// TwinCAT 3 PLC project AMKO_System
// Title: IBF_System
// Company: Industrial Brains B.V.
// ProjectVersion: 0.0.0.0
// Description: system and module base functions
// ProgramVersion: 3.1.4023.0
// libraries:
//   Device_Library, * (AMKO-Engineering)
//   HMI_Library, * (AMKO-Engineering)
//   Tc2_Standard, * (Beckhoff Automation GmbH)
//   Tc2_System, * (Beckhoff Automation GmbH)
//   Tc2_Utilities, * (Beckhoff Automation GmbH)
//   Tc3_Module, * (Beckhoff Automation GmbH)
//   Utilities_Library, * (AMKO-Engineering)
// project tree:
//   / PlcTask.TcTTO
//   FaultHandler/ Fb_SystemFaultHandler.TcPOU
//   GVLs/ GVL_Main.TcGVL
//   ModuleBase/Base/ Fb_ModuleBase.TcPOU
//   ModuleBase/DataTypes/ Udt_ModuleBase.TcDUT
//   SystemBase/DataTypes/ E_StateSystem.TcTLEO, Udt_ModuleId.TcDUT (not stored)
//   SystemBase/ SystemBase.TcPOU
//   _TESTS/ FB_DummyModule.TcPOU, PRG_TEST.TcPOU

CONFIGURATION AMKO_System
    RESOURCE PLC ON TwinCAT3
        TASK PlcTask(INTERVAL := T#10ms, PRIORITY := 20);
        PROGRAM SystemBase WITH PlcTask : SystemBase;
    END_RESOURCE
END_CONFIGURATION

// ---- ModuleBase/DataTypes/Udt_ModuleBase.TcDUT
TYPE Udt_ModuleBase :
STRUCT
	sModuleName 		: STRING := 'NA' 		; // Module name
	bModuleActive		: 	BOOL := FALSE 		; // Module is active in the system (will be ignored by system if false) 	
	// safety Inputs
	bEstopOk			:	BOOL ; // When estop is not ok, complete machine is shut down and reinitialization is required.
	bModuleSafetyOk		: 	BOOL ; // Module safety systems are ok and safe 
	bAirPressureOk		: 	BOOL ; // system safety condition monitorring air pressure ok
	bPowerSupplyOk		: 	BOOL ; // System power supply is ok
	// main system Inputs
	bCmdStart			: 	BOOL	:= FALSE ; // System start command 
	bCmdReset 			: 	BOOL	:= FALSE ; // reset all faults 
	bCmdPowerOff		:	BOOL	:= FALSE ; // power off module 
	bCmdStartManual 	: 	BOOL 	:= FALSE ; // Start up in manual mode
 	// Com to main system
	fbFaultHandler		: 	Fb_FaultHandler 		; // Fault handler 
	sStateIndicator		: 	STRING := ''			; // Operator message, indication of current step or function 

	// Fault indications
	bMissingCond	: BOOL := FALSE ; // Module missing condition active
	bFatalFault		: BOOL := FALSE ; // Module fatal fault is active
	bCycleFault		: BOOL := FALSE ; // Module cycle fault is active
	bOperatorWarning : BOOL := FALSE; //

	// State indication
	bIsSafe			: BOOL := FALSE ; // Module is safe and locked until safety is ok
	bNoreference	: BOOL := FALSE ; // Module Startup Undefined initialization required

	bInitializing	: BOOL := FALSE ; // Module startup initializing
	bInitialized	: BOOL := FALSE ; // Module startup initialized waiting for startup command

	bIdle 			: BOOL := FALSE ; // Module startup Idle no commands active

	bEnabling 		: BOOL := FALSE ; // Module Startup enabeling 
	bEnabled 		: BOOL := FALSE ; // Module Startup Enabled
	
	bHoming			: BOOL := FALSE ; // Module startup homing back to base position and recalibrate
	bHomed 			: BOOL := FALSE ; // Module startup homed waiting for further further commands

	bHolding 		: BOOL := FALSE ; // Module Module Hold motion command executing
	bHeld	 		: BOOL := FALSE ; // Module Hold Motion is held until command is released	
	
	bResetting 		: BOOL := FALSE ; // Module Reset resetting error status
	bResetDone 		: BOOL := FALSE ; // Module reset is done   

	bManual 		: BOOL := FALSE ; // Module Work status Module in Manual 
	bAutomatic 		: BOOL := FALSE ; // Module Work status Module in Automatic mode
	
	bPoweringOff	: BOOL := FALSE ; // Module is powering off
	bPoweredOff		: BOOL := FALSE ; // Module has powered off 	
	
	// manual functions 
	bDevicesAddedtoManual	: BOOL := FALSE ;
	bParametersAdded		: BOOL := FALSE ;
	// Persistent data
	bCmdWritePersistent  : BOOL := false ; // write persistent data to memory
END_STRUCT
END_TYPE

// ---- SystemBase/DataTypes/E_StateSystem.TcTLEO
{attribute 'qualified_only'}
{attribute 'strict'}
{attribute 'to_string'}
TYPE E_StateSystem :
(
	NoReference		, 	// system has not been initialized
	Initialize		, 	// System is initializing
	LoadParameters	, 	// System is loading parameters from/to file
	Safe			, 	// System is in safety state
	Enable			, 	// System is enabling 
	Home			, 	// system is hominig 
	Resetting		, 	// System is resetting
	Idle			, 	// system is waiting for commands
	Manual			, 	// System is in manual mode
	SemiAuto		, 	// System is in semi auto mode
	Automatic		, 	// system is in automatic mode 
	Fault			,	// System is in Fault state
	PowerOff		// system is powering off
)INT;
END_TYPE

// ---- GVLs/GVL_Main.TcGVL

{attribute 'qualified_only'} // Main system variables and state indicators
{attribute 'analysis':= '-33'}
VAR_GLOBAL CONSTANT
	cnMaxNUMBEROFMODULES 	: UDINT := 10 		; // "maximum" number of modules in the system
	CtAIRPRESSUREDELAY	: TIME 	:= T#500MS	; // Timout before air fault becomes active
	cbUPSPRESENT		: BOOL	:= FALSE 	; // Enable automatic shutdown when power is interupted
END_VAR
VAR_GLOBAL PERSISTENT
	nTotalUnitsProduced		: UDINT ; // Units produced 
END_VAR

// ---- SystemBase/SystemBase.TcPOU
{attribute 'reflection'}
PROGRAM SystemBase // system base program, from here all modules are controlled and the system functions are called.
VAR_INPUT // System configuration settings
	bIcfAirCheckPresent	: BOOL := TRUE; // System is not equiped with air pressure sensor 
END_VAR
VAR	// Fault indications
	bMissingCond		: BOOL := FALSE ; // Module missing condition active
	bFatalFault			: BOOL := FALSE ; // Module fatal fault is active
	bCycleFault			: BOOL := FALSE ; // Module cycle fault is active
	bOperatorWarning	: BOOL := FALSE ; // Module operator warning is active

	// Check values
	bReferenceOk		: BOOL := FALSE ; // All module references  have been checked

	// State indication
	bSafeStopping		: BOOL := FALSE ; // Module is stopping by safety
	bIsSafe				: BOOL := FALSE ; // Module is safe and locked until safety is ok
	bNoreference		: BOOL := FALSE ; // Module Startup Undefined initialization required

	bInitializing		: BOOL := FALSE ; // Module startup initializing
	bInitialized		: BOOL := FALSE ; // Module startup initialized waiting for startup command
	
	bParametersLoaded 	: BOOL := FALSE ; // Parameters have been loaded from the file(s) 

	bIdle 				: BOOL := FALSE ; // Module startup Idle no commands active

	bEnabling 			: BOOL := FALSE ; // Module Startup enabeling 
	bEnabled 			: BOOL := FALSE ; // Module Startup Enabled
	
	bHoming				: BOOL := FALSE ; // Module startup homing back to base position and recalibrate
	bHomed 				: BOOL := FALSE ; // Module startup homed waiting for further further commands

	bHolding 			: BOOL := FALSE ; // Module Module Hold motion command executing
	bHeld	 			: BOOL := FALSE ; // Module Hold Motion is held until command is released	
	
	bResetting 			: BOOL := FALSE ; // Module Reset resetting error status
	bResetDone 			: BOOL := FALSE ; // Module reset is done   

	bManual 			: BOOL := FALSE ; // Module Work status Module in Manual 
	
	bStartSemiAuto		: BOOL := FALSE ; // Start semi automatic mode 
	bSemiAuto			: BOOL := FALSE ; // Module work status module in semi automatic
	
	bStartAuto			: BOOL := FALSE ; // Start automatic mode
	bAutomatic 			: BOOL := FALSE ; // Module Work status Module in Automatic mode
	bStopAuto			: BOOL := FALSE ; // Start automatic mode
	bStoppingAuto		: BOOL := FALSE ; // Start automatic mode
	
	bCmdPause			: BOOL := FALSE ; // Pause all modules 
	bPaused 			: BOOL := FALSE ; // all modules are paused
	
	bPoweringOff		: BOOL := FALSE ; // Module is powering off
	bPoweredOff			: BOOL := FALSE ; // Module has powered off 	

	bModuleLocked		: BOOL := FALSE ; // a module is locked for commands
	
	bAckWarningsBusy	: BOOL := FALSE	; // The acknowledge process is busy
END_VAR
VAR
	// System inputs 
	ibPowerSupplyOk	 	AT%I*	: BOOL  ; // System Power supply is ok 
	iSystemSafetyFault	AT%I*	: BOOL	; // System safety Fault
	fbAirpressureOk 			: Fb_DevDigitalInputFunctions  	; // system airpressure is ok
	fbCmdResetSafety		 	: FB_DevPushbuttonLight 		; // System reset
	
	fTrigPowerSupply			: F_TRIG ; // falling edge trigger for power supply
	toffMainAir					: TOF	:= (PT := T#500MS ); // Main air supply off delay
	// System safety valve
	fbValveMainAirSupply		: FB_DevValve ; // Main air supply valve 
	
	// System HMI commands
	fbStartSemiAuto				: FB_DevHMIButton ; // HMI start semi automatic button 
	fbStartAuto					: FB_DevHMIButton ; // HMI start automatic button
	fbResetSystem				: FB_DevHMIButton ; // HMI Reset system
	fbCmdPowerOff				: FB_DevHMIButton ; // HMI Power off system
	fbAckWarning				: FB_DevHMIButton ; // HMI Acknowledge warnings

	// system Commands 
	fbCmdStartSystem		 	: FB_DevPushbuttonLight  		; // (re)start system input from button
	fbCmdStartAuto				: FB_DevPushbuttonLight			; // Start system automatic cycle
	fbCmdStopAuto				: FB_DevPushbuttonLight			; // Start system automatic cycle
	
	//System state
	bSafetyOK					: BOOL := FALSE ;
	bAirOk						: BOOL := FALSE ; // Air pressure is ok 
	bSystemOK					: BOOL := FALSE ; // all safety and vitals are OK
	eStateSystem				: E_StateSystem := E_StateSystem.NoReference ; // State of system
	// Set system variables
	fbSetSystemVariables		: Fb_SystemVariables ;
	
	// System Fault handling
	fbSystemFaultHandler		: Fb_SystemFaultHandler ;
	fbOperatorMessage			: FB_OperatorMessageDisplay ; //Operator message or system state message hadler 

	// Local Fault Handling
	fbFaultHandler				: Fb_FaultHandler 		; // Fault handler 
	stMessage					: UDT_Fault			; // Message data

 	// Module states
	nNumberOfModules			: UDINT := 0 ; // Number of modules added to the system 
	arpModules					: ARRAY [1..gvl_main.cnMaxNUMBEROFMODULES] OF Udt_ModuleId ; 

	// power down system function
	ntShutDown					: NT_Shutdown ; // shutdown system function 

	// Manual controller
	bDevicesAddedtoManual 		: BOOL := FALSE ; // Add system device (buttons) to manual controller
	

	// Function path 
	{attribute 'instance-path'} 
    {attribute 'noinit'}
	sPath			: STRING	; // Path name of function (used for manual reference
END_VAR
VAR // safety 
	// inputs 
	ibEstopOk 			AT%I*	: BOOL  ; // system emergency stop ok
	ibSystemSafetyOK	AT%I*	: BOOL  ; // System is safe 
	iSafetyFBErr		AT%I*	: BOOL	; // The "FB Error" group signal
	iSafetyComErr		AT%I*	: BOOL	; // The "Com Error" group signal
	iSafetyOtherErr		AT%I*	: BOOL	; // The "Other Err" group signal
	iSafetyOutErr		AT%I*	: BOOL	; // The "Out Err" group signal
	iSTOFault			AT%I* 	: BOOL	; // Motor safe torque off fault active
	
	// Outputs 
	qbSafetyErrAckn		AT%Q*	: BOOL ; // Safety error acknowledge
	qbRunSafety			AT%Q*	: BOOL ; // Run safety program
	qbResetSafety		AT%Q*	: BOOL ; // reset safety program
	qbSTOErrAckn		AT%Q*	: BOOL ; // Safet torque off error acnowledge

	// safety Reset Timer	
	TofSafetyErrAck				: TOF := (PT := T#500MS); // Safety reset timer
	TOfSTOErrAck				: TOF := (PT := T#500MS); // Safe torque off rest timer
END_VAR
VAR // Miscellaneous
	bFirstCycle : BOOL := TRUE; // Is this the first time the PRG is called?
	bPersistentDataFail	: BOOL := TRUE ;
END_VAR
VAR PERSISTENT // Persistent data check
	bPersistentFlag	: BOOL := FALSE ; // Persistent dat in tack flag
END_VAR

// Exec safety control
ExecSafetyControl();

// Call faulthandler
fbSystemFaultHandler( 	nNumberOfModules	:= nNumberOfModules,
						arpModules			:= arpModules,
						bsystemInitialized	:= bInitialized,
						bSystemFF			=> bFatalFault,
						bSystemCF			=> bCycleFault,
						bSystemMC			=> bMissingCond,
						bSystemOW			=> bOperatorWarning);

// Check if this is the first cycle the PRG is called
// if not, return. This is to make sure all modules are connected. 
IF bFirstCycle THEN
	bFirstCycle := FALSE;
	RETURN;
END_IF

// check system functions
IF bInitialized AND bParametersLoaded THEN 
	CheckSystemOK();
	CheckSystemCommands();
END_IF 

// Run system
ExecSystemRun();

// call device functions 
CallSystemFunctions();

// Call operator warning acknowledgement
ExecAckWarnings();

// Call modules 
CallModules();

METHOD PRIVATE CallModules : BOOL
VAR
	i : UDINT ;
END_VAR
VAR
	AllAutomatic : BOOL ;
	
	Stopping : BOOL;
	bAllStopped : BOOL;
END_VAR
// set base conditions
bReferenceOk	:= TRUE ;
bIsSafe			:= TRUE ;
bIdle			:= TRUE ;	
bHeld			:= TRUE ;
bResetDone 		S= bResetting	;
bManual			:= TRUE	;
bSemiAuto		:= TRUE ;
bAutomatic		:= FALSE; // Reverse feedback 
AllAutomatic 	:= TRUE ;
bStoppingAuto	:= TRUE ;
bEnabled		S= bEnabling ;
bPoweredOff		:= TRUE;
bHomed 			:= TRUE;
bPaused 		:= TRUE;
bAllStopped     := TRUE;

// copy inputs to modules 
FOR i := 1 TO nNumberOfModules DO 
	// set system commands
	arpModules[i].pFunction^.bEnable			:= bEnabled			;
	arpModules[i].pFunction^.bCmdReset			:= bResetting		;
	arpModules[i].pFunction^.bSafetyOK			:= NOT bSafeStopping;
	arpModules[i].pFunction^.bCmdPause			:= bCmdPause		; 
	// Read state indications 
	bReferenceOk 	:= arpModules[i].pFunction^.bReferenceOk 	AND bReferenceOk; 
	bIsSafe 		:= arpModules[i].pFunction^.bIsSafe 		AND bIsSafe		;
	bEnabled 		:= arpModules[i].pFunction^.bEnable 		AND bEnabled	;
	bHeld			:= arpModules[i].pFunction^.bHeld 			AND bHeld		;
	bResetDone		:= arpModules[i].pFunction^.bResetDone 		AND bResetDone	;
	bManual			:= arpModules[i].pFunction^.bManual 		AND bManual		;
	bSemiAuto		:= arpModules[i].pFunction^.bSemiAuto 		AND bSemiAuto	;
	bPoweredOff 		:= arpModules[i].pFunction^.bPoweredOff 		AND bPoweredOff	;
	bHomed			:= arpModules[i].pFunction^.bHomed			AND bHomed 		;
	bPaused			:= arpModules[i].pFunction^.bPaused			AND bPaused		;
	bModuleLocked	S= arpModules[i].pFunction^.bLocked							; // Module is locked for commnds
	bCmdPause 		R= arpModules[i].pFunction^.bReqContinue					; // Request continue from module
	bCmdPause		S= arpModules[i].pFunction^.bReqPause						; // Request for pause from module
	bAutomatic		S= arpModules[i].pFunction^.bAutomatic 						; // Stay in automatic even when one module is in automatic
	AllAutomatic	:= arpModules[i].pFunction^.bAutomatic 		AND AllAutomatic; // reset start automatic when al modules are in automatic operation
	bStoppingAuto	:= arpModules[i].pFunction^.bStopping 		AND bStoppingAuto; // reset start automatic when al modules are in automatic operation

	Stopping		:= arpModules[i].pFunction^.bStopping;
	
	bAllStopped     := NOT Stopping AND NOT bAutomatic AND bAllStopped;

	
END_FOR

// Reset start inputs
	bEnabling		R= bEnabled 	;
	bHolding		R= bHeld 		;
	bResetting		R= bResetDone 	;
	bStartSemiAuto	R= bSemiAuto	;
	bPoweringOff	R= bPoweredOff 	;
	bHoming			R= bHomed 		;
	bStartAuto		R= AllAutomatic	; 
	bStopAuto		R= bAllStopped	;
	bCmdPause		R= NOT bAutomatic	;
END_METHOD

METHOD PRIVATE CallSystemFunctions : BOOL
VAR_INPUT
END_VAR
// call parameter handler
GVL_Parameters.fbParameterHandler();
Device_Library.GVL_DevManual.fbManualControler();

// Execute button functions 
fbStartAuto		( 	tDelay			:= T#100MS,
					refFbManualCtrl	:= Device_Library.GVL_DevManual.fbManualControler,
					refFbFault 		:= fbFaultHandler );
fbStartSemiAuto ( 	tDelay			:= T#100MS,
					refFbManualCtrl	:= Device_Library.GVL_DevManual.fbManualControler,
					refFbFault 		:= fbFaultHandler ); 
fbResetSystem 	( 	Istatus			:= GVL_Message.bResetFaults,
					tDelay			:= T#5000MS,
					refFbManualCtrl	:= Device_Library.GVL_DevManual.fbManualControler,
					refFbFault 		:= fbFaultHandler ); 
fbAckWarning	(	Istatus			:= GVL_Message.bAckWarnings,
					tDelay			:= T#100MS,
					refFbManualCtrl := Device_Library.GVL_DevManual.fbManualControler,
					refFbFault 		:= fbFaultHandler );

fbCmdStartSystem(	refFbManualCtrl	:= Device_Library.GVL_DevManual.fbManualControler,
					refFbFault 		:= fbFaultHandler);
fbCmdStartAuto	(	refFbManualCtrl	:= Device_Library.GVL_DevManual.fbManualControler,
					refFbFault 		:= fbFaultHandler);
fbCmdStopAuto	(	refFbManualCtrl	:= Device_Library.GVL_DevManual.fbManualControler,
					refFbFault 		:= fbFaultHandler);

// execute input functions
fbValveMainAirSupply(	bEnable			:= TRUE,
						bSafetyOk		:= ibEstopOk,
						refFbManualCtrl	:= Device_Library.GVL_DevManual.fbManualControler,
						refFbFault 		:= fbFaultHandler);

// Add device functions to manual controller 
IF NOT bDevicesAddedtoManual THEN
	IF bIcfAirCheckPresent THEN
		Device_Library.GVL_DevManual.fbManualControler.CmdAddDevice( refToDevice := fbAirpressureOk 	);
	END_IF
	Device_Library.GVL_DevManual.fbManualControler.CmdAddDevice( refToDevice := fbCmdStartSystem	);
	Device_Library.GVL_DevManual.fbManualControler.CmdAddDevice( refToDevice := fbCmdStartAuto		);
	Device_Library.GVL_DevManual.fbManualControler.CmdAddDevice( refToDevice := fbCmdStopAuto		);
	Device_Library.GVL_DevManual.fbManualControler.CmdAddDevice( refToDevice := fbCmdResetSafety	);
	bDevicesAddedtoManual S= TRUE ;
END_IF
END_METHOD

METHOD INTERNAL CheckSystemCommands : BOOL
VAR_INPUT
END_VAR
// ===== full reset ======
	IF fbCmdResetSafety.bFcoDelay THEN 
		eStateSystem 	:= E_StateSystem.NoReference ;
	END_IF

// ====== power off ======
	IF fbCmdPowerOff.bFcoDelay THEN 
		eStateSystem := E_StateSystem.PowerOff ;
	END_IF
END_METHOD

METHOD PRIVATE CheckSystemOK : BOOL
// shutdown emediately if power is down 
fTrigPowerSupply(CLK := ibPowerSupplyOk);
ntShutDown(START := GVL_Main.cbUPSPRESENT AND (bPoweredOff OR fTrigPowerSupply.Q)); 

// ===== Check Air pressure =====
IF bIcfAirCheckPresent THEN
	fbAirpressureOk(refFbManualCtrl	:= Device_Library.GVL_DevManual.fbManualControler,
					refFbFault 		:= fbFaultHandler);
	bAirOk := fbAirpressureOk.bFcoDelay ;
ELSE
	bAirOk := TRUE ;
END_IF


// ===== Check if system is ok =====
	bSystemOK := TRUE ;
	bSystemOK := bAirOk 	AND bSystemOK ;
	bSystemOK := bSafetyOK	AND bSystemOK ;	
				
	IF NOT bSystemOK 
	AND eStateSystem > E_StateSystem.Safe 
	AND eStateSystem <> E_StateSystem.Resetting 
	THEN
		eStateSystem := E_StateSystem.Safe; 
	ELSIF (bFatalFault OR bCycleFault) 
	AND eStateSystem <> E_StateSystem.Resetting 
	THEN 
		eStateSystem := E_StateSystem.Fault ;
	END_IF

// ===== release system stop =====
bSafeStopping 	R= bIsSafe AND bSystemOK 		;
	
// ===== System messages ======
	IF NOT bAirOk THEN
		stMessage.Active 		:= TRUE ;
		stMessage.ComponentType	:= E_ComponentTypes.SafeIO ;
		stMessage.Discription	:= 'Main air Pressure low ';
		stMessage.LocationName	:= 'Main air supply';
		stMessage.LocationNumber:= 1;
		stMessage.FaultType		:= Utilities_Library.E_FaultTypes.FF;
		stMessage.MessageNumber	:= E_MessageNumbers.FF_Overload;
		stMessage.nModuleID		:= 0;
		GVL_HMI.bEstopActive 	:= TRUE ;
		GVL_HMI.sCmdEstopText 	:= 'AIR PRESSURE LOW';
	END_IF
	
// Main air control 
toffMainAir(IN := bSystemOK);
IF toffMainAir.Q THEN
	fbValveMainAirSupply.CmdOpen();
END_IF
END_METHOD

METHOD PUBLIC CmdAddModule : BOOL
VAR_INPUT
	refToModule : REFERENCE TO Fb_ModuleBase ; // reference to module function
END_VAR
VAR
	bModuleAdded	: BOOL := FALSE;
	i 				: UDINT ; 
END_VAR
// Check if device is not already in the array 
FOR i:= 1 TO GVL_Main.cnMaxNUMBEROFMODULES DO
	IF arpModules[i].pFunction = 0 THEN 
		nNumberOfModules:= i;
		EXIT;	
	ELSIF arpModules[i].sName = refToModule.sName THEN 
		bModuleAdded := TRUE ;
	END_IF 
END_FOR

// If device is not found add device to the list
IF NOT bModuleAdded AND nNumberOfModules >= 1 AND nNumberOfModules <= GVL_Main.cnMaxNUMBEROFMODULES THEN
	arpModules[nNumberOfModules].nNumber 	:= refToModule.nModuleID;
	arpModules[nNumberOfModules].sName		:= refToModule.sName	;
	arpModules[nNumberOfModules].pFunction 	:= ADR(refToModule)		;	
	bModuleAdded := TRUE ;
END_IF

CmdAddModule := bModuleAdded ;
END_METHOD

METHOD CmdReset : BOOL
VAR_INPUT
END_VAR
eStateSystem := E_StateSystem.Resetting;

CmdReset := TRUE;
END_METHOD

METHOD ExecAckWarnings : BOOL
VAR
	i : UDINT ;
END_VAR
//If required, run the acknowledge process 
IF (fbAckWarning.bFeStatus OR NOT bAckWarningsBusy) THEN
	bAckWarningsBusy := TRUE;
	
	FOR i := 1 TO nNumberOfModules DO 
		bAckWarningsBusy := arpModules[i].pFunction^.CmdAckOW() AND bAckWarningsBusy;
	END_FOR
END_IF
END_METHOD

METHOD PRIVATE ExecAutomatic : BOOL
VAR_INPUT
END_VAR
VAR
	i : UDINT ;
END_VAR
IF bStopAuto THEN 
	FOR i := 1 TO nNumberOfModules DO 
		arpModules[i].pFunction^.CmdStopAutomatic() ;
	END_FOR
ELSIF bStartAuto THEN 
	// Run automatic function in 
	FOR i := 1 TO nNumberOfModules DO 
		arpModules[i].pFunction^.CmdAutomatic() ;
	END_FOR
END_IF
	
ExecAutomatic := NOT bStartAuto;
END_METHOD

METHOD PRIVATE ExecHoming : BOOL
VAR_INPUT
END_VAR
VAR
	i : UDINT ;
END_VAR
// Home all modules
FOR i := 1 TO nNumberOfModules DO 
	IF NOT arpModules[i].pFunction^.bHomed THEN 
		arpModules[i].pFunction^.CmdHome();
	END_IF
END_FOR
 
ExecHoming := bHomed ;
END_METHOD

METHOD PUBLIC ExecManual : BOOL
VAR
	i : UDINT ;
END_VAR
bEnabled := FALSE ;
// Run automatic function in 
FOR i := 1 TO nNumberOfModules DO 
	arpModules[i].pFunction^.CmdManual() ;
END_FOR

ExecManual := bManual;
END_METHOD

METHOD PRIVATE ExecPowerOff : BOOL
VAR_INPUT
END_VAR
VAR 
	i : UDINT ;
END_VAR
// Power off all modules
FOR i := 1 TO nNumberOfModules DO 
	arpModules[i].pFunction^.CmdPowerOff () ;
END_FOR
 
ExecPowerOff := bPoweredOff ;
END_METHOD

METHOD PRIVATE ExecSafeHold : BOOL
VAR_INPUT
END_VAR
VAR
	i : UDINT ;
END_VAR
// Hold all modules
bStartAuto		:= FALSE;

FOR i := 1 TO nNumberOfModules DO 
	arpModules[i].pFunction^.CmdHold();
END_FOR

ExecSafeHold := bHeld ;
END_METHOD

METHOD PRIVATE ExecSafeReset : BOOL
VAR_INPUT
END_VAR
END_METHOD

METHOD PRIVATE ExecSafeStop : BOOL
VAR_INPUT
END_VAR
VAR
	i : UDINT ;
END_VAR
bSafeStopping 	S= NOT bIsSafe ;

bEnabling		:= FALSE;
bInitializing	:= FALSE;
bHoming			:= FALSE;
bStartAuto		:= FALSE;
bStartSemiAuto	:= FALSE;

// Module safe stop
IF bInitialized AND bReferenceOk THEN 
	FOR i := 1 TO nNumberOfModules DO 
		arpModules[i].pFunction^.CmdEstop();
	END_FOR
END_IF

IF bIsSafe THEN 
	fbValveMainAirSupply.CmdSafeStop();
END_IF
 
ExecSafeStop := bIsSafe ;
END_METHOD

METHOD PRIVATE ExecSafetyControl : BOOL
VAR_INPUT
END_VAR
IF ibEstopOk 
AND ibSystemSafetyOK
AND NOT iSTOFault
THEN
	bSafetyOK				S= TRUE ;
	GVL_HMI.bEstopActive 	:= FALSE ;
ELSE 
	bSafetyOK				:= FALSE ;
	GVL_HMI.bEstopActive 	:= TRUE ;
	IF eStateSystem > E_StateSystem.Safe 
	AND eStateSystem <> E_StateSystem.Resetting  THEN 
		eStateSystem			:= E_StateSystem.Safe ;
	END_IF
END_IF

// Set safety state and button light state
fbCmdResetSafety.bEnable S= TRUE ;
IF NOT ibEstopOk THEN 
	GVL_HMI.bEstopActive 	:= TRUE ;
	fbCmdResetSafety.CmdOn() ;
ELSIF NOT ibSystemSafetyOK OR iSTOFault THEN 
	fbCmdResetSafety.CmdBlinkSlow() ;
ELSIF NOT bAirOk OR NOT bSystemOK THEN
	fbCmdResetSafety.CmdBlinkFast() ;
END_IF



// Safety reset button function
fbCmdResetSafety(	tDelay			:= T#30S ,
					refFbManualCtrl	:= Device_Library.GVL_DevManual.fbManualControler,
					refFbFault 		:= fbFaultHandler); 

// Link Safetty Reset
qbResetSafety := fbCmdResetSafety.bFeStatus AND NOT bSafetyOK ;

// Set safety system in run mode
IF NOT iSafetyFBErr 
AND NOT iSafetyComErr
AND NOT iSafetyOtherErr
AND NOT iSafetyOutErr
AND NOT iSystemSafetyFault 
AND bInitialized THEN 
	qbRunSafety := TRUE ;
ELSE 
	qbRunSafety := FALSE;
END_IF

// reset safety faults
TofSafetyErrAck	(IN := qbSafetyErrAckn	);
TOfSTOErrAck	(IN := qbSTOErrAckn 	);
qbSTOErrAckn	:= FALSE ;
qbSafetyErrAckn := FALSE ;

IF iSafetyFBErr THEN 
	GVL_HMI.sCmdEstopText 	:= 'Safety Program Function block error';
	IF NOT qbRunSafety AND NOT TofSafetyErrAck.Q THEN 
		qbSafetyErrAckn := TRUE; 
	END_IF
	stMessage.Active := TRUE ;
	stMessage.ComponentType	:= E_ComponentTypes.SafeIO ;
	stMessage.Discription	:= 'Safety program is in fault state.';
	stMessage.LocationName	:= 'Main safety';
	stMessage.LocationNumber:= 1;
	stMessage.FaultType		:= Utilities_Library.E_FaultTypes.FF;
	stMessage.MessageNumber	:= E_MessageNumbers.FF_Unknown;
	stMessage.nModuleID		:= 0;
	GVL_HMI.sCmdEstopText 	:= 'Safety program is in fault state.';
ELSIF iSafetyComErr THEN
	GVL_HMI.sCmdEstopText 	:= 'Safety program com error';
	IF NOT qbRunSafety AND NOT TofSafetyErrAck.Q THEN 
		qbSafetyErrAckn := TRUE ;
	END_IF
	stMessage.Active 		:= TRUE ;
	stMessage.ComponentType	:= E_ComponentTypes.SafeIO ;
	stMessage.Discription	:= 'Emergency stop fault, check emergency button wiring ';
	stMessage.LocationName	:= 'Emergency stop safety';
	stMessage.LocationNumber:= 1;
	stMessage.FaultType		:= Utilities_Library.E_FaultTypes.FF;
	stMessage.MessageNumber	:= E_MessageNumbers.FF_Unknown;
	stMessage.nModuleID		:= 0;
	GVL_HMI.sCmdEstopText 	:= 'Emergency stop fault, check emergency button wiring ';
ELSIF iSafetyOutErr THEN
	GVL_HMI.sCmdEstopText 	:= 'Safety program out error';
	IF NOT qbRunSafety AND NOT TofSafetyErrAck.Q THEN 
		qbSafetyErrAckn := TRUE ;
	END_IF
	stMessage.Active 		:= TRUE ;
	stMessage.ComponentType	:= E_ComponentTypes.SafeIO ;
	stMessage.Discription	:= 'Emergency stop fault, check wiring ';
	stMessage.LocationName	:= 'Emergency stop safety';
	stMessage.LocationNumber:= 1;
	stMessage.FaultType		:= Utilities_Library.E_FaultTypes.FF;
	stMessage.MessageNumber	:= E_MessageNumbers.FF_Unknown;
	stMessage.nModuleID		:= 0;
	GVL_HMI.sCmdEstopText 	:= 'Emergency stop fault, check wiring ';
ELSIF iSafetyOtherErr THEN
	GVL_HMI.sCmdEstopText 	:= 'Safety program other error';
	IF NOT qbRunSafety AND NOT TofSafetyErrAck.Q THEN 
		qbSafetyErrAckn := TRUE ;
	END_IF
	stMessage.Active 		:= TRUE ;
	stMessage.ComponentType	:= E_ComponentTypes.SafeIO ;
	stMessage.Discription	:= 'Safety program is in fault state. ';
	stMessage.LocationName	:= 'Emergency stop safety';
	stMessage.LocationNumber:= 1;
	stMessage.FaultType		:= Utilities_Library.E_FaultTypes.FF;
	stMessage.MessageNumber	:= E_MessageNumbers.FF_Unknown;
	stMessage.nModuleID		:= 0;
	GVL_HMI.sCmdEstopText 	:= 'Safety program is in fault state. ';
ELSIF iSystemSafetyFault THEN
// System safety function faults 
	GVL_HMI.sCmdEstopText 	:= 'Collision detection Fault check sensor wiring';
	IF NOT qbRunSafety AND NOT TofSafetyErrAck.Q THEN 
		qbSafetyErrAckn := TRUE ;
	END_IF
	stMessage.Active 		:= TRUE ;
	stMessage.ComponentType	:= E_ComponentTypes.SafeIO ;
	stMessage.Discription	:= 'Collision safety fault, check collision detection wiring ';
	stMessage.LocationName	:= 'Collision safety';
	stMessage.LocationNumber:= 1;
	stMessage.FaultType		:= Utilities_Library.E_FaultTypes.FF;
	stMessage.MessageNumber	:= E_MessageNumbers.FF_Unknown;
	stMessage.nModuleID		:= 0;
	GVL_HMI.sCmdEstopText 	:= 'System safety fault, check wiring ';
ELSIF iSTOFault THEN
	GVL_HMI.sCmdEstopText 	:= 'Motor safety fault';
	qbSTOErrAckn 			:= Sys_Variables.HeartBeat ;
	stMessage.Active 		:= TRUE ;
	stMessage.ComponentType	:= E_ComponentTypes.SafeIO ;
	stMessage.Discription	:= 'Collision safety fault, check collision detection wiring ';
	stMessage.LocationName	:= 'Collision safety';
	stMessage.LocationNumber:= 1;
	stMessage.FaultType		:= Utilities_Library.E_FaultTypes.FF;
	stMessage.MessageNumber	:= E_MessageNumbers.FF_Unknown;
	stMessage.nModuleID		:= 0;
	GVL_HMI.sCmdEstopText 	:= 'Motor safe torque off fault';
ELSIF NOT ibEstopOk THEN
	GVL_HMI.sCmdEstopText 	:= 'Emergency stop pressed';
ELSIF NOT ibSystemSafetyOK THEN 
	GVL_HMI.sCmdEstopText 	:= 'Safety bumper pressed';
END_IF
END_METHOD

METHOD PUBLIC ExecSemiAuto : BOOL
VAR
	i : UDINT ;
END_VAR
// Run automatic function in 
FOR i := 1 TO nNumberOfModules DO 
	arpModules[i].pFunction^.CmdSemiAuto() ;
END_FOR

ExecSemiAuto := bSemiAuto;
END_METHOD

METHOD INTERNAL ExecSystemRun : BOOL
VAR_INPUT
END_VAR
// set system variables 
fbSetSystemVariables();

// State machine 
CASE eStateSystem OF 
	E_StateSystem.NoReference:
		// Reset HMI state
		HMI_Library.GVL_HMI.bCmdSemiAuto 	:= FALSE;
		HMI_Library.GVL_HMI.bCmdAutomatic	:= FALSE;
		HMI_Library.GVL_HMI.bCmdSettings	:= FALSE;
		HMI_Library.GVL_HMI.bCmdManual		:= FALSE;
		HMI_Library.GVL_HMI.bCmdParemeter	:= FALSE;
		HMI_Library.GVL_HMI.eShownScreen	:= E_BaseVisu.Idle;
		bHomed			:= FALSE ;
		bEnabled		:= FALSE ;
		IF bReferenceOk THEN
			eStateSystem 	:= E_StateSystem.Initialize ;
		END_IF
	E_StateSystem.Initialize:
		IF Init() THEN
			eStateSystem := E_StateSystem.LoadParameters	;
		END_IF
	E_StateSystem.LoadParameters:
		bParametersLoaded := GVL_Parameters.fbParameterHandler.Init(); 
		IF bParametersLoaded THEN
			eStateSystem := E_StateSystem.Safe ;
		ELSIF GVL_Parameters.fbParameterHandler.bError THEN 
			eStateSystem := E_StateSystem.NoReference ;
		END_IF
	E_StateSystem.Safe:
		IF bIsSafe 
		AND bSystemOK THEN 
			IF bFatalFault OR bCycleFault THEN
				eStateSystem := E_StateSystem.Fault ;
			ELSE
				eStateSystem 	:= E_StateSystem.Enable;
			END_IF
		ELSIF fbResetSystem.bFeStatus THEN
			eStateSystem	:= E_StateSystem.Resetting;
		ELSE 
			ExecSafeStop();
		END_IF
	E_StateSystem.Enable:
		bEnabling 	:= bSystemOK;
		IF GVL_HMI.bCmdManual THEN
			eStateSystem := E_StateSystem.Manual ;
		ELSIF bEnabled THEN 
			fbCmdStartSystem.CmdBlinkFast();
			IF fbCmdResetSafety.bFeStatus THEN
				eStateSystem := E_StateSystem.Resetting ;
			ELSIF fbCmdStartSystem.bFeStatus THEN
				eStateSystem := E_StateSystem.Home ;
			END_IF
		END_IF
	E_StateSystem.Home:	
		IF fbCmdResetSafety.bFeStatus THEN
			eStateSystem := E_StateSystem.Safe;			
		ELSIF ExecHoming() THEN
			eStateSystem := E_StateSystem.Idle;
		END_IF
	E_StateSystem.Resetting:
		IF NOT bResetDone THEN 
			bResetting S= TRUE ;
		ELSIF NOT bSafetyOK THEN 
			eStateSystem := E_StateSystem.Safe ;
		ELSIF bFatalFault OR bCycleFault THEN
			eStateSystem := E_StateSystem.Fault ;
		ELSIF bHomed THEN
			eStateSystem := E_StateSystem.Idle ;
		ELSE 
			eStateSystem := E_StateSystem.Enable ;
		END_IF
	E_StateSystem.Idle:
		fbCmdStartSystem.CmdBlinkSlow();
		IF fbCmdResetSafety.bFeStatus OR fbResetSystem.bFeStatus THEN
			eStateSystem := E_StateSystem.Resetting;			
		ELSIF GVL_HMI.bCmdManual THEN 
			eStateSystem := E_StateSystem.Manual ;
		ELSIF bSystemOK AND fbCmdStartSystem.bFeStatus THEN 
			eStateSystem := E_StateSystem.SemiAuto ;
		END_IF
	E_StateSystem.Manual:
		IF fbCmdResetSafety.bFeStatus THEN
			eStateSystem := E_StateSystem.Safe;			
		ELSIF Device_Library.GVL_DevManual.bManualModeActive THEN
			ExecManual();
		END_IF
		
		IF NOT GVL_HMI.bCmdManual THEN
			EStateSystem := E_StateSystem.Enable;
		END_IF 
	E_StateSystem.SemiAuto:
		ExecSemiAuto();
		GVL_HMI.bCmdSemiAuto 	:= TRUE;
		IF fbCmdResetSafety.bFeStatus THEN
			eStateSystem := E_StateSystem.Idle;			
		ELSIF (fbCmdStartAuto.bFeStatus 
		OR fbStartAuto.bFcoDelay 
		OR bAutomatic)
		AND NOT bModuleLocked THEN 
			bStartAuto 		:= TRUE ;
			bStopAuto 		:= FALSE;
			eStateSystem 	:= E_StateSystem.Automatic ;
		END_IF					
	E_StateSystem.Automatic:
		ExecAutomatic();
		Gvl_HMI.bCmdAutomatic := TRUE;
		IF fbCmdResetSafety.bFeStatus THEN
			eStateSystem := E_StateSystem.Safe;
		ELSIF bAutomatic THEN
			IF fbCmdStartSystem.bFeStatus THEN
				eStateSystem := E_StateSystem.Idle ;
			ELSIF fbCmdStopAuto.bFeStatus THEN
				bStopAuto := TRUE;
			ELSIF fbCmdStartAuto.bFeStatus OR bMissingCond THEN  
				bCmdPause 	:= NOT bPaused ;
			END_IF
		ELSIF NOT bStartAuto AND NOT bStopAuto THEN 
			eStateSystem := E_StateSystem.SemiAuto ;
		END_IF
		
		// Start button light control
		IF bAutomatic THEN 
			fbCmdStartAuto.CmdOn();
		ELSE
			fbCmdStartAuto.CmdBlinkFast(); 				
		END_IF
	E_StateSystem.Fault:
		IF fbResetSystem.bFeStatus OR fbCmdResetSafety.bFeStatus THEN
			bResetDone		:= FALSE ;
			eStateSystem 	:= E_StateSystem.Resetting ;
		ELSIF bFatalFault THEN 
			ExecSafeStop();
		ELSIF bCycleFault THEN 
			ExecSafeHold();	
		END_IF 
	E_StateSystem.PowerOff:
		ExecPowerOff();
	ELSE 
		;		
END_CASE

bModuleLocked := FALSE ;
END_METHOD

METHOD PRIVATE Init : BOOL
VAR_INPUT
END_VAR
VAR
	i : UDINT ;
END_VAR
// initialize system functions
IF bIcfAirCheckPresent THEN
	fbAirpressureOk.Init	( 	nId 		:= 1,
								nParentId	:= 0 );
END_IF 

fbCmdResetSafety.Init	(	nId 		:= 2,
							nParentId	:= 0 );

fbValveMainAirSupply.Init(	nId			:= 3,
							nParentId	:= 0,
							eResetState	:= E_ValveResetState.Res_Closed,
							eSafeState	:= E_ValveResetState.Res_Closed);

fbCmdStartSystem.Init	( 	nId 		:= 4,
							nParentId	:= 0 );

fbCmdStartAuto.Init		( 	nId 		:= 5,
							nParentId	:= 0 );

fbCmdStopAuto.Init		( 	nId 		:= 6,
							nParentId	:= 0 );
							
// Initialize all modules
bInitialized	:= TRUE ;
FOR i := 1 TO nNumberOfModules DO 
	IF NOT arpModules[i].pFunction^.bInitialized THEN 
		arpModules[i].pFunction^.CmdInit();
	END_IF
	bInitialized 	:= bInitialized AND arpModules[i].pFunction^.bInitialized;
	bInitializing 	:= NOT bInitialized ;
	// Set feedback to screen (needs to be added)
 END_FOR
 
 Init := bInitialized ;
END_METHOD

END_PROGRAM

// ---- FaultHandler/Fb_SystemFaultHandler.TcPOU
FUNCTION_BLOCK INTERNAL Fb_SystemFaultHandler
VAR_INPUT
	nNumberOfModules	: UDINT := 0; // Number of modules connected to the system fault handler
	bsystemInitialized	: BOOL 	; // System init is done
END_VAR
VAR_IN_OUT
	arpModules			: ARRAY [1..gvl_main.cnMaxNUMBEROFMODULES] OF Udt_ModuleId ;
END_VAR
VAR_OUTPUT
	// Fault types 
	bSystemFF			: BOOL 	:= FALSE	; // System fatal fault is active
	bSystemCF			: BOOL 	:= FALSE	; // System Cycle fault is active
	bSystemMC 			: BOOL 	:= FALSE	; // a missing condition is active only 
	bSystemOW			: BOOL	:= FALSE	; // A operator warning is active
END_VAR
VAR
	// Message variables
	bCmdSnoozeMessage	: REFERENCE TO BOOL  	:= GVL_Message.bCmdSnoozeMessage; // Snooze message display
	arActiveFaults 		: REFERENCE TO ARRAY [0..Param_Messages.nMAX_MESSAGES_SHOWN] OF UDT_Fault := GVL_Message.arActiveFaults ; // Active faults overview for showing in HMI
	arOldFaults 		: ARRAY [0..Param_Messages.nMAX_MESSAGES_SHOWN] OF UDT_Fault ; // Old faults overview for comparing to active
	arWriteToLog		: ARRAY [0..Param_Messages.nMAX_MESSAGES_SHOWN] OF UDT_Fault ; // Fault array for writing to log file 
	// Message logging
	dToday				: DATE 	; 
	nWriteStep			: UDINT := 0 ;
	bWriteError			: BOOL 	; // write to file error occured
	nWriteErroId		: UDINT ; // write error id
	// Write variables
	sActFileName		: STRING;
	hFile				: UINT	:= 0;(* File handle of the source file *)
	sMessageString		: ARRAY [0..Param_Messages.nMESSAGE_COLUMNS] OF STRING (GVL_Parameters.MAX_CSV_FIELD_LENGTH); (* temporary parameter buffer to string*)
	sCSVLine			: T_MaxString := '';(* Single CSV text line (row, record), we are using string as record buffer (your are able to see created fields) *)
	sCSVField			: T_MaxString := '';(* Single CSV field value (column, record field) *)
END_VAR
VAR // functions 
	tofSnoozeMessages	: TOF ; // timer function for message snoozing
	// Log to file functions
	fbFileOpen		: FB_FileOpen	;(* Opens file *)
	fbFileClose		: FB_FileClose	;(* Closes file *)
	fbFileGets		: FB_FileGets	;(* Reads one record (line) *)
	fbFilePuts		: FB_FilePuts	;(* Writes one record (line) *)
	fbReader		: FB_CSVMemBufferReader;(* Helper function block used to parse CSV data bytes (single record line) *)
	fbWriter		: FB_CSVMemBufferWriter;(* Helper function block used to create CSV data bytes (single record line) *)
END_VAR 
VAR CONSTANT
	stEmptyMessageUdt : UDT_Fault := (	Active 			:= FALSE,
									FaultType 		:= E_FaultTypes.NA,
									MessageNumber	:= 0,
									LocationNumber	:= 0,
									Discription 	:= '',
									LocationName	:= '',
									ComponentType	:= E_ComponentTypes.NA,
									StartTime		:= DT#2020-1-1-00:00:00,
									EndTime			:= DT#2020-1-1-00:00:00,
									FullFaultId		:= '0'	)  ;
END_VAR

IF nNumberOfModules > 0 THEN 
	// Check modules for active messages 
	CheckForModuleFaults();
END_IF

IF bsystemInitialized THEN
	// set system fault bits 
	ExecSetFaultBit(); 
	// Log faults when they are reset
	ExecMessageCompare();
	// Logfile writer 
	ExecWriteToLog();
END_IF

// Message Screen controller 
ExecScreenControl();

METHOD PRIVATE CheckForModuleFaults : BOOL // check all modules for faults and copy them to the main fault array
VAR
	// functional variables
	i 					: UDINT ;
	j 					: UDINT ;
	// temporary fault storage
	arTempFaults	: ARRAY [0..Param_Messages.nMAX_MESSAGES_SHOWN] OF UDT_Fault ; // internal fault array
	p				: UDINT	;
END_VAR
{warning disable C0371}
IF NOT __ISVALIDREF(arpModules) THEN
	RETURN;
END_IF

// Go over modules to check for fault messages 
FOR i := 1 TO nNumberOfModules DO 
	// Check for active messages
	FOR j := 0 TO Param_Messages.nMAX_MESSAGES_SHOWN DO
		IF arpModules[i].pFunction^.fbFaultHandler.arActiveFaults[j].FaultType <> E_FaultTypes.NA THEN 
			arTempFaults[p]:= arpModules[i].pFunction^.fbFaultHandler.arActiveFaults[j] ;
			p := MIN( p + 1, Param_Messages.nMAX_MESSAGES_SHOWN);
		ELSE
			EXIT ;
		END_IF
	END_FOR
END_FOR

arOldFaults		:= arActiveFaults 	;
arActiveFaults	:= arTempFaults 	;
{warning restore C0371}
END_METHOD

METHOD PRIVATE ExecMessageCompare : BOOL
VAR
	// functional variables
	i 			: UDINT ;
	j 			: UDINT ;
	bFaultFound : BOOL ;
	p			: UDINT;
END_VAR
// Check if any changes occured in the active faults
FOR i := 0 TO Param_Messages.nMAX_MESSAGES_SHOWN DO
	// break loop if fault is empty
	IF  arOldFaults[i].FaultType = E_FaultTypes.NA THEN  
		EXIT;
	ELSE
		// check if the fault is still active
		bFaultFound := FALSE; 
		FOR j := 0 TO Utilities_Library.Param_Messages.nMAX_MESSAGES_SHOWN DO
			IF arOldFaults[i].FullFaultId = arActiveFaults[j].FullFaultId THEN
				bFaultFound := TRUE;
				EXIT;
			END_IF
		END_FOR
		// if the fault is not faund then wrtie it to the logging array for loging
		IF NOT bFaultFound THEN 
			arWriteToLog[p] := arOldFaults[i] ;
			p := p + 1 ; 
		END_IF
	END_IF
END_FOR

ExecSortMessages();
END_METHOD

METHOD PRIVATE ExecScreenControl : BOOL // Control message screen 
VAR_INPUT
END_VAR
tofSnoozeMessages(IN := bCmdSnoozeMessage, PT := GVL_Message.tMESSAGESNOOZEDURATION);

// Set screen control 
IF bSystemCF OR bSystemFF THEN 
	GVL_Message.bHideFaults := FALSE ;
	GVL_Message.bHideReset	:= FALSE ; 
ELSIF bSystemOW THEN
	GVL_Message.bHideWarnAck := FALSE;
ELSIF bSystemMC AND NOT tofSnoozeMessages.Q THEN 
	GVL_Message.bHideFaults := FALSE ;
ELSE
	GVL_Message.bHideFaults := TRUE ;
	GVL_Message.bHideReset	:= TRUE ; 
	GVL_Message.bHideWarnAck:= TRUE ;
END_IF
END_METHOD

METHOD PRIVATE ExecSetFaultBit : BOOL
VAR
	// functional variables
	i 			: UDINT ;
END_VAR
bSystemFF	:= FALSE ;
bSystemCF	:= FALSE ;
bSystemMC	:= FALSE ;
bSystemOW	:= FALSE ;

FOR i := 0 TO Param_Messages.nMAX_MESSAGES_SHOWN DO
	bSystemFF	:= arActiveFaults[i].FaultType = E_FaultTypes.FF OR bSystemFF;
	bSystemCF	:= arActiveFaults[i].FaultType = E_FaultTypes.CF OR bSystemCF;
	bSystemMC	:= arActiveFaults[i].FaultType = E_FaultTypes.MC OR bSystemMC;
	bSystemOW   := arActiveFaults[i].FaultType = E_FaultTypes.OW OR bSystemOW;
END_FOR
END_METHOD

METHOD INTERNAL ExecSortMessages : BOOL
VAR
	i : UDINT ;
	k : UDINT ;
	stTempMessageStorage : UDT_Fault ; // Temporary message storage for sorting
END_VAR
FOR k := 1 TO Param_Messages.nMAX_MESSAGES_SHOWN - 1 DO 
	FOR i := 0 TO Param_Messages.nMAX_MESSAGES_SHOWN - 2 DO 
		IF arActiveFaults[i].FaultType < arActiveFaults[i+1].FaultType THEN 
			stTempMessageStorage 	:= arActiveFaults[i];
			arActiveFaults[i]		:= arActiveFaults[i+1];
			arActiveFaults[i+1]		:= stTempMessageStorage;
		END_IF
	END_FOR	 
END_FOR

ExecSortMessages := TRUE;
END_METHOD

METHOD PRIVATE ExecWriteToLog : BOOL
VAR 
	i : UDINT ; 
	p : UDINT ; // Fault array pointer
END_VAR
dToday := DT_TO_DATE(Sys_Variables.SystemTime);
// create file name with Current date 
sActFileName 	:= CONCAT(STR1 := Param_Messages.sLOGFILE_PATH	, STR2 := Param_Messages.sLOGFILE_NAME	);
sActFileName 	:= CONCAT(STR1 := sActFileName					, STR2 := DATE_TO_STRING(dToday)		);
sActFileName 	:= CONCAT(STR1 := sActFileName					, STR2 := '.csv'						);

// ===== Start file write =====
CASE nWriteStep OF
	0:	(* Wait until log array is filled *)
		IF arWriteToLog[0].FaultType <> E_FaultTypes.NA THEN 
			hFile				:= 0;
			nWriteStep 			:= 1;
		ELSE 
			RETURN ;
		END_IF
	1:	(* Open source file *)
		fbFileOpen(  bExecute := FALSE  );
		fbFileOpen( sNetId := GVL_Parameters.sNetId, sPathName := sActFileName , nMode := FOPEN_MODEAPPEND OR FOPEN_MODETEXT,(* Open file in TEXT mode! *)
					ePath := PATH_GENERIC, bExecute := TRUE );
		nWriteStep := nWriteStep + 1 ;
	2:(* Wait until open not busy *)
		fbFileOpen( bExecute := FALSE, bError => bWriteError, nErrID => nWriteErroId, hFile => hFile );
		IF NOT fbFileOpen.bBusy THEN
			IF NOT fbFileOpen.bError THEN
				nWriteStep := nWriteStep + 1 ;
			ELSE(* Error: file not found? *)
				nWriteStep := 100;
			END_IF
		END_IF
	3: (* Check if faultrecord is active if so skip record *)
		nWriteStep := nWriteStep + 1 ;
	4:(* Convert one PLC record to CSV format *)
		sCSVLine := '';
		fbWriter.eCmd := eEnumCmd_First;(* Write first field value *)
		// write message data to string
		sMessageString[0] 	:= TO_STRING(arWriteToLog[p].FaultType				);
		sMessageString[1]	:= DT_TO_STRING(arWriteToLog[p].StartTime			);
		sMessageString[2]	:= DT_TO_STRING(Sys_Variables.SystemTime			);
		sMessageString[3]	:= UDINT_TO_STRING(arWriteToLog[p].MessageNumber	);
		sMessageString[4]	:= UDINT_TO_STRING(arWriteToLog[p].LocationNumber	); 
		sMessageString[5]	:= arWriteToLog[p].Discription						;
		sMessageString[6]	:= arWriteToLog[p].LocationName						;
		sMessageString[7]	:= TO_STRING(arWriteToLog[p].ComponentType			);
		// write data to .csv buffer 
		FOR i := 0 TO Param_Messages.nMESSAGE_COLUMNS BY 1 DO
			sCSVField := STRING_TO_CSVFIELD(in :=  sMessageString[i], FALSE );
			(* Add new field to the record buffer *)
			fbWriter( 	pBuffer := ADR( sCSVLine ), cbBuffer := SIZEOF( sCSVLine ) - 1, putValue := sCSVField, pValue := 0, cbValue := 0,
						bCRLF := ( i = Param_Messages.nMESSAGE_COLUMNS ) );(* bCRLF == TRUE => Write CRLF after the last field value *)
			IF fbWriter.bOk THEN
				fbWriter.eCmd := eEnumCmd_Next;
			ELSE
				nWriteStep := 100;
				RETURN;
			END_IF
		END_FOR(* FOR nColumn := 0... *)

		(* FB_FilePuts adds allready CR (carriage return) to the written line.
		We have to replace the $R$L characters with $L character to avoid double CR. *)
		IF RIGHT( sCSVLine, 2 ) = '$R$L' THEN
			sCSVLine := REPLACE( sCSVLine, '$L', 2, LEN( sCSVLine ) - 1 );
		END_IF
		nWriteStep := nWriteStep + 1 ;
	5:	(* Write single text line to file *)
		fbFilePuts( bExecute := FALSE );
		fbFilePuts( sNetId := GVL_Parameters.sNetId, hFile := hFile, sLine := sCSVLine, bExecute := TRUE );
		nWriteStep := nWriteStep + 1 ;
	6:(* Wait until write not busy *)
		fbFilePuts( bExecute := FALSE, bError => bWriteError, nErrID => nWriteErroId );
		IF NOT fbFilePuts.bBusy THEN
			IF NOT fbFilePuts.bError THEN
				nWriteStep := nWriteStep + 1 ;
			ELSE(* Error *)
				nWriteStep := 100;
			END_IF
		END_IF
	7: (* clear fault from array and go to next fault *)
		arWriteToLog[p]:= stEmptyMessageUdt;
		IF p < Param_Messages.nMAX_MESSAGES_SHOWN THEN 
			p := p +1 ;
		END_IF
		nWriteStep := nWriteStep +1 ;
	8: (* If fault is active then repeat previous step, else close file*)		
		IF  arWriteToLog[p].FaultType <> E_FaultTypes.NA THEN 
			nWriteStep := 3 ;
		ELSE
			nWriteStep := 10;
		END_IF
	10:	(* Close source file *)
		fbFileClose( bExecute := FALSE );
		fbFileClose( sNetId := GVL_Parameters.sNetId, hFile := hFile, bExecute := TRUE );
		nWriteStep := 11;
	11:(* Wait until close not busy *)
		fbFileClose( bExecute := FALSE, bError => bWriteError, nErrID => nWriteErroId );
		IF ( NOT fbFileClose.bBusy ) THEN
			hFile 		:= 0;
			nWriteStep 	:= 100;
		END_IF
	100: (* Error or ready nWriteStep => cleanup *)
		IF ( hFile <> 0 ) THEN
			nWriteStep	:= 10; (* Close the source file *)
		ELSE
			nWriteStep 	:= 0;	(* Ready *)
			ExecWriteToLog := TRUE ;
		END_IF
END_CASE
END_METHOD

END_FUNCTION_BLOCK

// ---- ModuleBase/Base/Fb_ModuleBase.TcPOU
{attribute 'reflection'}
FUNCTION_BLOCK PUBLIC ABSTRACT Fb_ModuleBase
VAR_INPUT
	nModuleID			: 	UDINT 	:= 1 	; // module reference number used for fault, enable, reset, and safety functions (default := 1, 0 = main system)
	// main system Inputs
	bEnable				: 	BOOL	:= FALSE ; // (autolinked) module enable 	
	bCmdReset 			: 	BOOL	:= FALSE ; // (AutoLinked) reset all faults 
	bSysFatalFault		: 	BOOL 	:= FALSE ; // (AutoLinked) System fatal fault active
	bSysCycleFault		: 	BOOL 	:= FALSE ; // (AutoLinked) System fatal fault active 
	bCmdPause			: 	BOOL 	:= FALSE ; // Pause command	bCmdToStart			
	// Internal safety 
	bSafetyOK			: BOOL := FALSE ; // Module internal safety is ok
END_VAR
VAR_OUTPUT
	sName 				: STRING 	:= 'NA' 			; // Module name
	bAddedToSystem		: BOOL 		:= FALSE 			; // module has been added to the system
 	// Com to main system
	fbFaultHandler		: 	Fb_FaultHandler 		; // Fault handler 
	sStateIndicator		: 	STRING := ''			; // Operator message, indication of current step or function 

	// Fault indications
	bMissingCond	: BOOL := FALSE ; // Module missing condition active
	bFatalFault		: BOOL := FALSE ; // Module fatal fault is active
	bCycleFault		: BOOL := FALSE ; // Module cycle fault is active
	bReqPause		: BOOL := FALSE ; // Request for auto cycle pause
	bReqContinue	: BOOL := FALSE ; // Request for auto cycel continue
	// Check values
	bReferenceOk	: BOOL := FALSE ; // All module references  have been checked
	// State indication
	bIsSafe			: BOOL := FALSE ; // Module is safe and locked until safety is ok
	bNoreference	: BOOL := FALSE ; // Module Startup Undefined initialization required
	bInitialized	: BOOL := FALSE ; // Module startup initialized waiting for startup command
	bHomed 			: BOOL := FALSE ; // Module startup homed waiting for further further commands

	bHolding 		: BOOL := FALSE ; // Module Module Hold motion command executing
	bHeld	 		: BOOL := FALSE ; // Module Hold Motion is held until command is released	
	
	bResetDone 		: BOOL := FALSE ; // Module reset is done   
	bCmdAckOW		: BOOL := FALSE	; // Acknowledge the operator warning
	bAckOWDone		: BOOL := FALSE	; // The operator warning is acknowledged
	
	bManual 		: BOOL := FALSE ; // Module Work status Module in Manual
	bSemiAuto		: BOOL := FALSE ; // Module work status in semi automatic
	bStartAuto		: BOOL := FALSE ; // Module start automatic cycle 
	bAutomatic 		: BOOL := FALSE ; // Module Work status Module in Automatic mode
	bPaused			: BOOL := FALSE ; // Module paused
	bStopAuto		: BOOL := FALSE ; // Module Stop automatic
	bStopping		: BOOL := FALSE ; // MOdule stopping auto cycle
	
	bPoweringOff	: BOOL := FALSE ; // Module is powering off
	bPowerdOff		: BOOL := FALSE ; // Module has powerd off 	

	bLocked			: BOOL := FALSE ; // module is locked for commands
END_VAR
VAR 
	// Internal functions 
	ReCmdReset 			: R_TRIG ;
	TofResetCmd			: TOF ;
	// manual functions 
	bParametersAdded	: BOOL := FALSE ;
	// Persistent data
	bCmdWritePersistent : BOOL := FALSE ; // write persistent data to memory
	// Module data
	stMessage			: UDT_Fault			; // Message data
	// Function path 
	{attribute 'instance-path'} 
    {attribute 'noinit'}
	sPath				: STRING	; // Path name of function (used for manual reference)
END_VAR

// Get device name from function
IF sName = 'NA' THEN 
	sName := F_FBNameFromPath(sPath := sPath);
END_IF

// Add module to system
IF NOT bAddedToSystem THEN
	bAddedToSystem S= SystemBase.CmdAddModule(refToModule := THIS^);
	RETURN;
END_IF

IF NOT bReferenceOk THEN 
	bReferenceOk S= CheckReferences();
	RETURN;
ELSE 
	// Execute functions
	ExecMainBaseFunctions();
	SetCycles();
END_IF

// Reset pause request 
bReqPause 		R= bPaused ;
bReqContinue    R= NOT bPaused 	;

METHOD PROTECTED ABSTRACT CallComponents : BOOL
VAR_INPUT
END_VAR
END_METHOD

METHOD PROTECTED ABSTRACT CheckCollision : BOOL // Checks device commands for positble collisions  and block if necesarry
VAR_INPUT
END_VAR
END_METHOD

METHOD PUBLIC CheckReferences : BOOL
VAR_INPUT
END_VAR
bReferenceOk := TRUE;
END_METHOD

METHOD INTERNAL CmdAckOW : BOOL
VAR_INPUT
END_VAR
bCmdAckOW := TRUE;

CmdAckOW := bAckOWDone;
END_METHOD

METHOD INTERNAL CmdAutomatic : BOOL
VAR_INPUT
END_VAR
IF NOT bAutomatic THEN 
	bStartAuto 		:= TRUE ;
	bStopping		:= FALSE;
END_IF 

CmdAutomatic 	:= bAutomatic;
END_METHOD

METHOD INTERNAL CmdEstop : BOOL
VAR_INPUT
END_VAR
ExecSafeStop();
bSemiAuto		:= FALSE ;
bAutomatic 		:= FALSE ;

CmdEstop := bIsSafe ;
END_METHOD

METHOD INTERNAL CmdHold : BOOL
VAR_INPUT
END_VAR
ExecHold();


CmdHold := bHeld ;
END_METHOD

METHOD Internal CmdHome : BOOL
VAR_INPUT
END_VAR
ExecHome();

CmdHome := bHomed;
END_METHOD

METHOD INTERNAL CmdInit : BOOL
VAR_INPUT
END_VAR
ExecInit();

CmdInit := bInitialized;
END_METHOD

METHOD Internal CmdManual : BOOL
VAR_INPUT
END_VAR
ExecManual();

CmdManual := bManual;
END_METHOD

METHOD INTERNAL CmdPowerOff : BOOL
VAR_INPUT
END_VAR
ExecPowerOff();
bAutomatic := FALSE ;

CmdPowerOff := bPowerdOff;
END_METHOD

METHOD INTERNAL CmdSemiAuto : BOOL
VAR_INPUT
END_VAR
ExecSemiAuto();

CmdSemiAuto := bSemiAuto ;
END_METHOD

METHOD INTERNAL CmdStopAutomatic : BOOL
VAR_INPUT
END_VAR
IF bAutomatic THEN 
	bStartAuto 		:= FALSE ;
	bStopAuto 		:= TRUE ;
END_IF 

CmdStopAutomatic 	:= NOT bAutomatic;
END_METHOD

METHOD PROTECTED ABSTRACT ExecAutomatic : BOOL
VAR_INPUT
END_VAR
END_METHOD

METHOD PUBLIC ExecBaseFunctions : BOOL
VAR_INPUT
END_VAR
END_METHOD

METHOD ExecFaultHandling : BOOL
VAR_INPUT
END_VAR
// Call message function
	fbFaultHandler();
	fbFaultHandler.CmdAddFault( stFault := stMessage );

	bFatalFault := fbFaultHandler.bActFF ;
	bCycleFault := fbFaultHandler.bActCF ;
	
	IF bFatalFault THEN
		ExecSafeStop()	;
	ELSIF bCycleFault THEN
		bHeld			S= ExecHold();
		bHolding 		:= NOT bHeld ;
	END_IF

// Call reset functions
	ReCmdReset( CLK := bCmdReset);
	
	IF ReCmdReset.Q THEN 
		bResetDone := FALSE ;
	ELSIF NOT bResetDone THEN 
		IF bInitialized THEN
			bResetDone := ExecReset() AND fbFaultHandler.CmdReset();
		ELSE
			bResetDone := TRUE ;		
		END_IF
	END_IF
	
	bCmdReset := FALSE ;


	
// Reset safe state when enable is active
	bIsSafe R= bSafetyOK ;

// Prevent automatic start when fault is active
	bStartAuto R= bCmdReset OR bFatalFault OR bCycleFault ;
	bStopAuto  R= bCmdReset OR bFatalFault OR bCycleFault ;
END_METHOD

METHOD PROTECTED ABSTRACT ExecHold : BOOL
VAR_INPUT
END_VAR
END_METHOD

METHOD PROTECTED ABSTRACT ExecHome : BOOL
VAR_INPUT
END_VAR
END_METHOD

METHOD PROTECTED ABSTRACT ExecInit : BOOL
VAR_INPUT
END_VAR
END_METHOD

METHOD INTERNAL ExecMainBaseFunctions : BOOL
VAR_INPUT
END_VAR
// Call fault handling function 
ExecFaultHandling();

//Handle the operator warning acknowledgement
IF (bCmdAckOW) THEN
	bAckOWDone := ExecOWAck();
ELSE
	bAckOWDone := FALSE;
END_IF;

//Reset Operator warning acknowledgement command bit
bCmdAckOW := FALSE;

// Check for any Internal collisions
IF bInitialized THEN
	CheckCollision();
END_IF

// Call components 
CallComponents();

// Run automatic function 
IF bStopAuto OR bStopping THEN 
	bStopping 	:= ExecAutomatic();
	bAutomatic  := FALSE;
	bStopAuto	:= FALSE;
	bStartAuto 	:= FALSE;
	bSemiAuto	:= FALSE;
ELSIF bStartAuto OR bAutomatic THEN 
	bAutomatic 	:= ExecAutomatic();
	bStartAuto 	:= FALSE;
	bSemiAuto	:= FALSE;
ELSIF bEnable AND NOT bAutomatic AND NOT bStopping THEN
	bAutomatic 	:= FALSE;
	bSemiAuto  	:= ExecSemiAuto();
ELSE
	bStopping   := FALSE;
	bAutomatic 	:= FALSE;
	bSemiAuto	:= FALSE;
END_IF

// Run Base Functions 
IF bInitialized 
AND bEnable
AND bHomed 
AND NOT bManual THEN 
	ExecBaseFunctions();
END_IF

// Persistent data 
IF bCmdWritePersistent THEN 
	bCmdWritePersistent R= DataManager.FbPersistentManager.Write();
END_IF
END_METHOD

METHOD PROTECTED ExecManual : BOOL
VAR_INPUT
END_VAR
bManual := true;
END_METHOD

METHOD PROTECTED ExecOWAck : BOOL
VAR_INPUT
END_VAR
//A helper method to prevent modules that don't use the operator warning
//to have to handle the acknowledgement
ExecOWAck := bCmdAckOW;
END_METHOD

METHOD PROTECTED ABSTRACT ExecPowerOff : BOOL
VAR_INPUT
END_VAR
END_METHOD

METHOD PROTECTED ABSTRACT ExecReset : BOOL
VAR_INPUT
END_VAR
END_METHOD

METHOD PROTECTED ABSTRACT ExecSafeStop : BOOL
VAR_INPUT
END_VAR
END_METHOD

METHOD PROTECTED ABSTRACT ExecSemiAuto : BOOL
VAR_INPUT
END_VAR
END_METHOD

METHOD PROTECTED SetCycles : BOOL
VAR_INPUT
END_VAR
SetCycles := true ;
END_METHOD

END_FUNCTION_BLOCK

// ---- _TESTS/FB_DummyModule.TcPOU
FUNCTION_BLOCK FB_DummyModule EXTENDS Fb_ModuleBase
VAR_INPUT
END_VAR
VAR_OUTPUT
END_VAR
VAR
END_VAR

SUPER^();

METHOD PROTECTED  CallComponents : BOOL
VAR_INPUT
END_VAR
END_METHOD

METHOD PROTECTED  CheckCollision : BOOL // Checks device commands for positble collisions  and block if necesarry
VAR_INPUT
END_VAR
END_METHOD

METHOD PROTECTED  ExecAutomatic : BOOL
VAR_INPUT
END_VAR
bAutomatic := TRUE;
ExecAutomatic := bAutomatic;
END_METHOD

METHOD PROTECTED  ExecHold : BOOL
VAR_INPUT
END_VAR
bHeld := TRUE;
END_METHOD

METHOD PROTECTED  ExecHome : BOOL
VAR_INPUT
END_VAR
bHomed := TRUE;
END_METHOD

METHOD PROTECTED  ExecInit : BOOL
VAR_INPUT
END_VAR
bInitialized := TRUE;
END_METHOD

METHOD PROTECTED  ExecPowerOff : BOOL
VAR_INPUT
END_VAR
bPowerdOff := TRUE;
END_METHOD

METHOD PROTECTED  ExecReset : BOOL
VAR_INPUT
END_VAR
bResetDone := TRUE;
END_METHOD

METHOD PROTECTED  ExecSafeStop : BOOL
VAR_INPUT
END_VAR
bIsSafe := TRUE;
END_METHOD

METHOD PROTECTED  ExecSemiAuto : BOOL
VAR_INPUT
END_VAR
bSemiAuto := TRUE;
END_METHOD

END_FUNCTION_BLOCK

// ---- _TESTS/PRG_TEST.TcPOU
PROGRAM PRG_TEST
VAR
	fbDummyModule : FB_DummyModule;
END_VAR

(*
CONTAINS CODE NEEDED FOR AUTOMATIC TESTING
*)

// SystemBase is the master program. it controls all underlying modules.
SystemBase();

// Call modules
fbDummyModule(nModuleID:= 1);

// HMI control
// GVL_HMI.fbHMIControl();

END_PROGRAM
